FUNCTION_BLOCK OperatorLogical (* Template for an empty basic function block *)
  (* Standard: 61499-2; Description: Copyright (c) 2019 Jan Holzweber This program and the accompanying materials are made available under the terms of the Eclipse Public License 2.0 which is available at https://www.eclipse.org/legal/epl-2.0/ SPDX-License-Identifier: EPL-2.0 *)
  (* Version 1.0, 2019-06-05, jholz *)
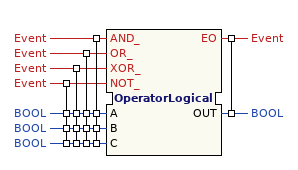
  EVENT_INPUT
    AND_ WITH A, B, C;
    OR_ WITH A, B, C;
    XOR_ WITH A, B, C;
    NOT_ WITH A, B, C;
  END_EVENT
  EVENT_OUTPUT
    EO WITH OUT;
  END_EVENT
  VAR_INPUT
    A : BOOL;
    B : BOOL;
    C : BOOL;
  END_VAR
  VAR_OUTPUT
    OUT : BOOL;
  END_VAR
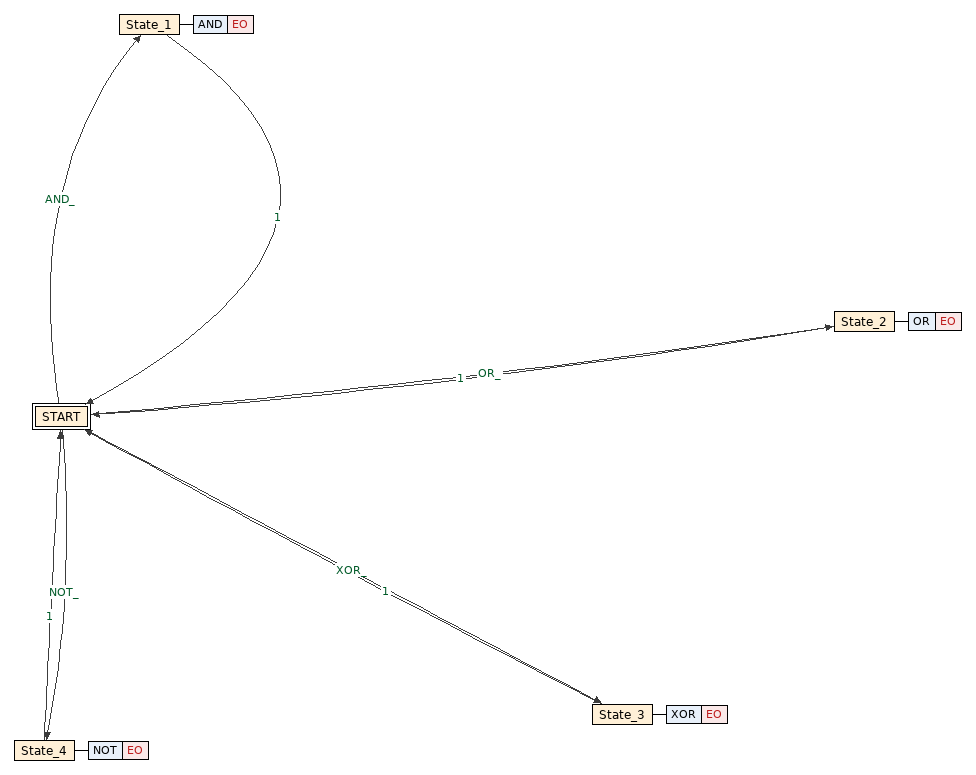
  EC_STATES
    START; (* Initial State *)
    State_1 : AND -> EO;
    State_2 : OR -> EO;
    State_3 : XOR -> EO;
    State_4 : NOT -> EO;
  END_STATES
  EC_TRANSITIONS
    State_1 TO START := 1;
    START TO State_1 := AND_;
    START TO State_2 := OR_;
    START TO State_3 := XOR_;
    START TO State_4 := NOT_;
    State_4 TO START := 1;
    State_3 TO START := 1;
    State_2 TO START := 1;
  END_TRANSITIONS
  ALGORITHM AND IN ST: (* new algorithm *)
OUT:=A and B and C;
  END_ALGORITHM
  ALGORITHM OR IN ST: (* new algorithm *)
OUT:=A or B or C ;
  END_ALGORITHM
  ALGORITHM XOR IN ST: (* new algorithm *)
OUT:=A XOR B XOR C;
  END_ALGORITHM
  ALGORITHM NOT IN ST: (* new algorithm *)
OUT:=NOT A;
  END_ALGORITHM
END_FUNCTION_BLOCK
